# EPICS substitutions: parser/test/test2.substitutions
file "test.template" {
    pattern {TEST}
    {ETT}
}
